FUNCTION_BLOCK FB_WORD_BCD_TO_INT (* Convert 4 BCD digits to INT *)
  (* Standard: 61499-1; Classification: Simple FB; Function: BCD conversion; Type: WORD to INT *)
  (* Version 0.0, 2007-08-27, JHC, Holobloc Inc *)
  (* Compiler header: package fb.rt.math; *)
  (* Compiler classdef: SimpleFB *)
  (* Compiler Java Sun JDK 1.6.0 *)
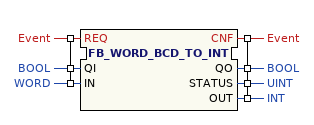
  EVENT_INPUT
    REQ WITH QI, IN; (* Normal Execution Request *)
  END_EVENT
  EVENT_OUTPUT
    CNF WITH QO, STATUS, OUT; (* Execution Confirmation *)
  END_EVENT
  VAR_INPUT
    QI : BOOL; (* Input event qualifier *)
    IN : WORD; (* 4 BCD digits *)
  END_VAR
  VAR_OUTPUT
    QO : BOOL; (* Output event qualifier *)
    STATUS : UINT; (* 0=OK, 2=conversion error per 61499-1 Table D.1 *)
    OUT : INT; (* Converted value of IN *)
  END_VAR
  ALGORITHM REQ IN Java: (* Normally executed algorithm *)
QO.value=QI.value;
STATUS.value = 0;
if(!QO.value){
STATUS.value = 1;
 return;}
int result = 0;
int temp = IN.value;
int digit = 0;
for (int i=0; i<4; i++){
temp = temp <<<4;
digit = temp & 15;
if(digit>9){
QO.value = false;
STATUS.value = 2;
return;
}
result = result*10+digit;
}
}
  END_ALGORITHM
END_FUNCTION_BLOCK
